(* Schneider Machine Expert - Basic project ATG, file version 2.6.0.0 *)
(* CompanyInformations: Name=PT. Yerry Primatama Hosindo [Engineering Div], Street=Jl. Raya Serpong Km. 99 Blok GN No. 09-10, City=Gunung Sindur, Bogor, ZipCode=16340, Country=Indonesia, WebSite=www.yerryprimatama-engineering.com *)
(* ProjectInformations: Name=Automatic Tank Gauging, Description=********Disclaimer Of Warranty********
THE INFORMATION CONTAINED HEREIN IS PROVIDED "AS IS" WITHOUT WARRANTIES OF ANY KIND, EITHER EXPRESS OR IMPLIED, INCLUDING WITHOUT LIMITATION, ALL IMPLIED WARRANTIES OF MERCHANTABILITY, FITNESS FOR A PARTICULAR PURPOSE, NON-INFRINGEMENT OR OTHER VIOLATION OF RIGHTS. SCHNEIDER ELECTRIC DOES NOT WARRANT OR MAKE ANY REPRESENTATIONS REGARDING THE USE, VALIDITY, ACCURACY, OR RELIABILITY OF, OR THE RESULTS OF THE USE OF, OR OTHERWISE, RESPECTING THE MATERIALS, SPECIFICATIONS, CHARACTERISTICS OR OTHER INFORMATION SPECIFIED HEREIN. FURTHERMORE, ALL WARRANTIES, CONDITIONS, REPRESENTATIONS, INDEMNITIES AND GUARANTEES WITH RESPECT TO THE ACCURACY, OPERATION, CAPACITY, SPEED, FUNCTIONALITY, QUALIFICATIONS, OR CAPABILITIES OF THE SOFTWARE, SYSTEMS AND SERVICES COMPRISING OR UTILIZED IN THE COURSE OF APPLYING THIS INFORMATION, SPECIFICATIONS, OR MATERIALS, WHETHER EXPRESS OR IMPLIED, ARISING BY LAW, CUSTOM, PRIOR ORAL OR WRITTEN STATEMENTS BY SCHNEIDER ELECTRIC, OR OTHERWISE (INCLUDING, BUT NOT LIMITED TO ANY WARRANTY OF SATISFACTORY QUALITY, MERCHANTABILITY, FITNESS FOR PARTICULAR PURPOSE, TITLE AND NON-INFRINGEMENT) ARE HEREBY EXPRESSLY EXCLUDED AND DISCLAIMED:
********Disclaimer Of Liability*********
UNDER NO CIRCUMSTANCES (INCLUDING NEGLIGENCE OR FORESEEABLE MISUSE) WILL SCHNEIDER ELECTRIC BE LIABLE FOR ANY DIRECT, INDIRECT, SPECIAL, INCIDENTAL, PUNITIVE OR CONSEQUENTIAL DAMAGES (INCLUDING WITHOUT LIMITATION, BUSINESS INTERRUPTION, DELAYS, LOSS OF DATA OR PROFIT) ARISING OUT OF THE APPLICATION OF THE INFORMATION, SPECIFICATIONS, CHARACTERISTICS OR MATERIALS CONTAINED HEREIN EVEN IF SCHNEIDER ELECTRIC HAS BEEN ADVISED OF THE POSSIBILITY OF SUCH DAMAGES.
************************************
The information, program and configuration contained herein are provided as general training on the products concerned, in part, by way of theoretical and/or hypothetical examples.  Only you, the user, can be aware of all the conditions and factors present during setup, operation, and maintenance of your machine and its application; therefore, only you, the user, can determine the automation equipment and the related safeties and interlocks which can be properly used.  When selecting automation and control equipment and related software for a particular application, you must refer to the applicable local and national standards and regulations.
************************************
Copyright © 2021 PT. Yerry Primatama Hosindo [ Engineering Division]. All rights reserved. *)
(* UserInformations: LastName=Firmansyah, FirstName=Ahmad Fauzi, CellNumber=+62 822 3222 2862, Email=ahmad.fauzi@yerryprimatama.com, Street=Taman Bougenville, Jl. Jelidro Tama No. E4, City=Surabaya, ZipCode=60217, Country=Indonesia *)

HARDWARE
  Cpu 0: TM221CE16R
  ModuleExtensionObject 0: TM2AMM6HT
  EthernetConfiguration: NetworkName=M221, IpAllocationMode=FixedAddress, IpAddress=192.168.0.21, SubnetMask=255.255.255.0
  SerialLineConfiguration: Baud=Baud115200, Parity=ParityEven, DataBits=DataBits8, StopBits=StopBits1, PhysicalMedium=PhysicalMediumRs485, TransmissionMode=TransmissionModeModbusRtu, SlaveId=1, Addressing=SlaveAddressing
  MastTask: UsePeriodScanMode=false, PeriodScan=100
  FastTask: Period=255
  CpuBehavior: StartingMode=StartAsPreviousState, AutoSaveRamOnEeprom=true, WatchdogPeriod=250

SYMBOLS  (address, symbol, comment, settings)
  %MW0      PRODUCT_HEIGHT
  %MW1      WATER_HEIGHT
  %MW2      TEMPERATURE
  %MF12     VOLUME_MM
  %MF14     PRODUCT_VOLUME
  %MF18     WATER_VOLUME
  %MF20     VOLUME_MAX
  %MF22     PRODUCT_ULLAGE
  %MF26     ACT_TEMPERATURE
  %MF28     IN_WATER_HIGH
  %MF30     IN_PRODUCT_HIGH
  %MF32     IN_PRODUCT_LOW
  %MF34     VCF
  %MF36     VOLUME15
  %Q0.0     WATER_HIGH
  %Q0.1     PRODUCT_HIGH
  %Q0.2     PRODUCT_LOW
  %IW1.0    PRD_HEIGHT  [Type=Type_4_20mA_Fast, Scope=Scope_Customized, Minimum=0, Maximum=5000]
  %IW1.1    WTR_HEIGHT  [Type=Type_4_20mA_Fast, Scope=Scope_Customized, Minimum=0, Maximum=5000]
  %IW1.2    TEMP  [Type=Type_4_20mA_Fast, Scope=Scope_Customized, Minimum=0, Maximum=1000]

POU Tank-01
  (* SectionNumber=1 *)

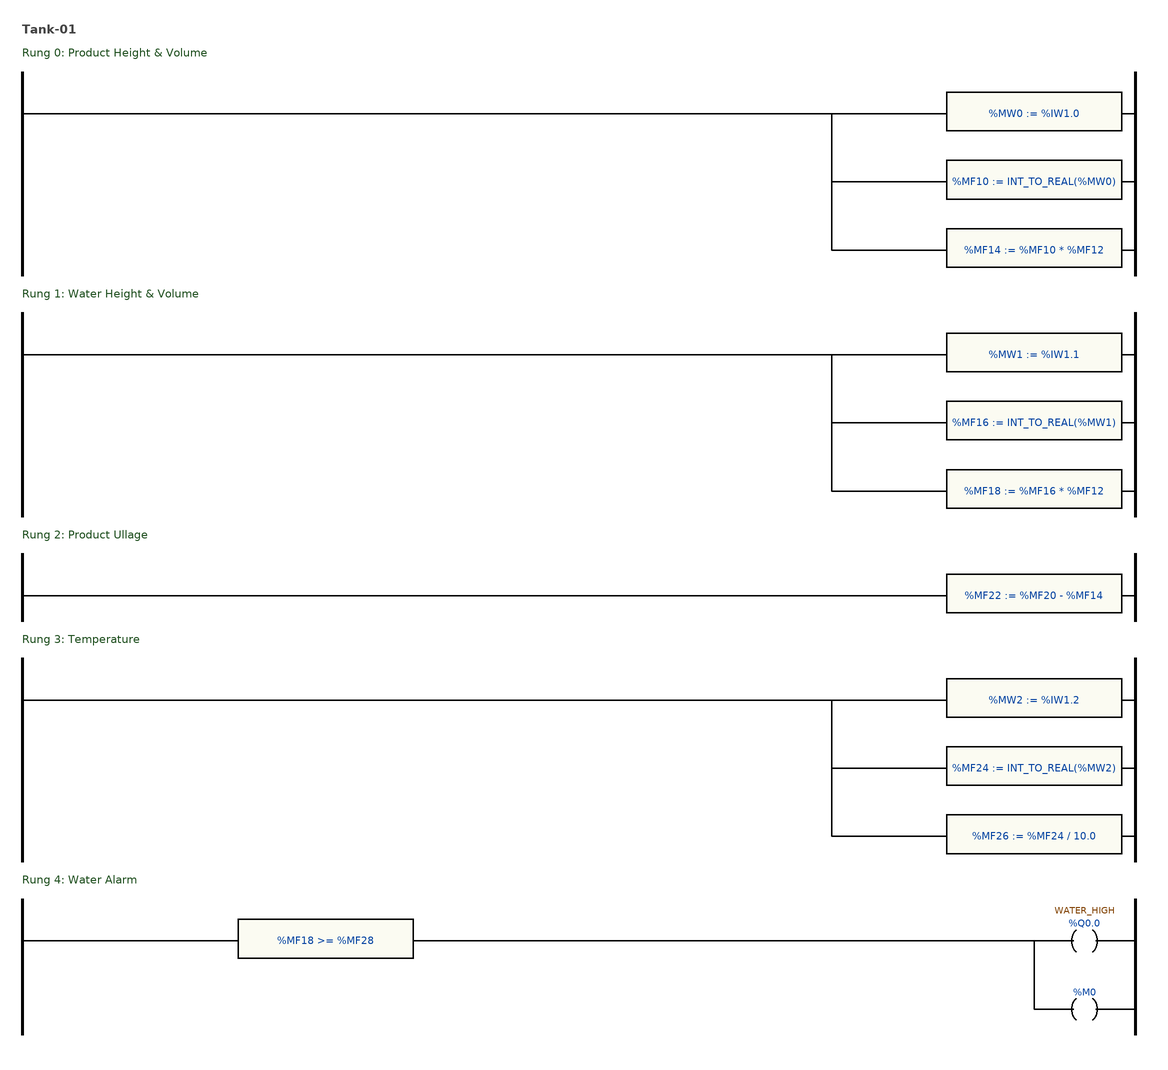

// Rung 0: Product Height & Volume
  LD 1
  [ %MW0 := %IW1.0 ]      (* PRODUCT_HEIGHT, PRD_HEIGHT *)
  [ %MF10 := INT_TO_REAL ( %MW0 ) ](* PRODUCT_HEIGHT *)
  [ %MF14 := %MF10 * %MF12 ](* PRODUCT_VOLUME, VOLUME_MM *)
  // as ST:
  //   PRODUCT_HEIGHT := PRD_HEIGHT;
  //   %MF10 := INT_TO_REAL ( PRODUCT_HEIGHT );
  //   PRODUCT_VOLUME := %MF10 * VOLUME_MM;

// Rung 1: Water Height & Volume
  LD 1
  [ %MW1 := %IW1.1 ]      (* WATER_HEIGHT, WTR_HEIGHT *)
  [ %MF16 := INT_TO_REAL ( %MW1 ) ](* WATER_HEIGHT *)
  [ %MF18 := %MF16 * %MF12 ](* WATER_VOLUME, VOLUME_MM *)
  // as ST:
  //   WATER_HEIGHT := WTR_HEIGHT;
  //   %MF16 := INT_TO_REAL ( WATER_HEIGHT );
  //   WATER_VOLUME := %MF16 * VOLUME_MM;

// Rung 2: Product Ullage
  LD 1
  [ %MF22 := %MF20 - %MF14 ](* PRODUCT_ULLAGE, VOLUME_MAX, PRODUCT_VOLUME *)
  // as ST:
  //   PRODUCT_ULLAGE := VOLUME_MAX - PRODUCT_VOLUME;

// Rung 3: Temperature
  LD 1
  [ %MW2 := %IW1.2 ]      (* TEMPERATURE, TEMP *)
  [ %MF24 := INT_TO_REAL ( %MW2 ) ](* TEMPERATURE *)
  [ %MF26 := %MF24 / 10.0 ](* ACT_TEMPERATURE *)
  // as ST:
  //   TEMPERATURE := TEMP;
  //   %MF24 := INT_TO_REAL ( TEMPERATURE );
  //   ACT_TEMPERATURE := %MF24 / 10.0;

// Rung 4: Water Alarm
  LD [ %MF18 >= %MF28 ]   (* WATER_VOLUME, IN_WATER_HIGH *)
  ST %Q0.0                (* WATER_HIGH *)
  ST %M0
  // as ST:
  //   WATER_HIGH := WATER_VOLUME >= IN_WATER_HIGH;
  //   %M0 := WATER_VOLUME >= IN_WATER_HIGH;

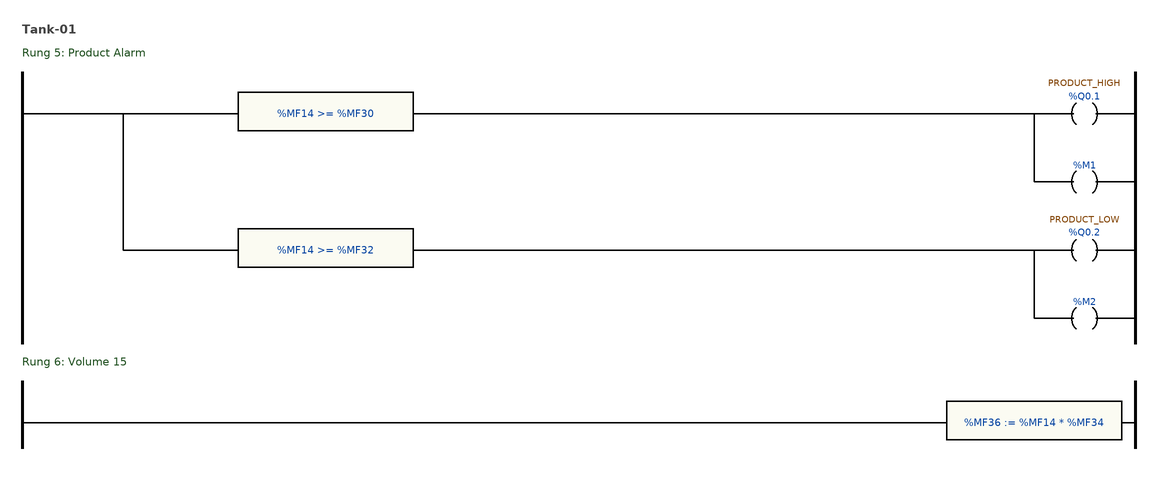

// Rung 5: Product Alarm
  LD 1
  MPS
  AND [ %MF14 >= %MF30 ]  (* PRODUCT_VOLUME, IN_PRODUCT_HIGH *)
  ST %Q0.1                (* PRODUCT_HIGH *)
  ST %M1
  MPP
  AND [ %MF14 >= %MF32 ]  (* PRODUCT_VOLUME, IN_PRODUCT_LOW *)
  ST %Q0.2                (* PRODUCT_LOW *)
  ST %M2
  // as ST:
  //   PRODUCT_HIGH := PRODUCT_VOLUME >= IN_PRODUCT_HIGH;
  //   %M1 := PRODUCT_VOLUME >= IN_PRODUCT_HIGH;
  //   PRODUCT_LOW := PRODUCT_VOLUME >= IN_PRODUCT_LOW;
  //   %M2 := PRODUCT_VOLUME >= IN_PRODUCT_LOW;

// Rung 6: Volume 15
  LD 1
  [ %MF36 := %MF14 * %MF34 ](* VOLUME15, PRODUCT_VOLUME, VCF *)
  // as ST:
  //   VOLUME15 := PRODUCT_VOLUME * VCF;
